(* PLC project CoDeSys External Library Template, WAGO e!COCKPIT e!COCKPIT, author 3S - Smart Software Solutions GmbH *)
(* stored: creationDateTime 2019-10-29T12:22:40.6298767, version 3.5.5.30, modificationDateTime 2019-10-24T14:40:07.960949, organization 3S - Smart Software Solutions GmbH *)
(* Library project template with all possible element types, docu and a sample project structure *)

FUNCTION_BLOCK fbFiltrWartoscAnalogowa
  VAR_INPUT
    rWartoscWejsciowa : REAL;
    rWartoscWejsciowaZaraportowana : REAL;
    rDeadband : REAL;
    tCzasMinimalny : TIME := TIME#5s0ms;
    tCzasMaksymalny : TIME := TIME#1m0s0ms;
    rWynikMnoznik : REAL := 1;
    rWynikOffset : REAL := 0;
  END_VAR
  VAR_OUTPUT
    rWartoscWyjsciowa : REAL;
  END_VAR
  VAR
    rWartoscWejsciowaZaraportowanaReferencja : REAL;
    fbCzasMinimalny : TON;
    fbCzasMaksymalny : TON;
    xCzasMinimalny : BOOL;
    xCzasMaksymalny : BOOL;
  END_VAR

            xCzasMinimalny := TRUE;
xCzasMaksymalny := TRUE;	

IF rWartoscWejsciowaZaraportowana <> rWartoscWejsciowaZaraportowanaReferencja THEN
	rWartoscWejsciowaZaraportowanaReferencja := rWartoscWejsciowaZaraportowana;
	xCzasMinimalny := FALSE;
	xCzasMaksymalny := FALSE;	
END_IF

IF fbCzasMinimalny.Q AND ABS(rWartoscWyjsciowa - (rWartoscWejsciowa * rWynikMnoznik + rWynikOffset)) > rDeadband THEN
	rWartoscWyjsciowa := rWartoscWejsciowa * rWynikMnoznik + rWynikOffset;
	xCzasMinimalny := FALSE;
	xCzasMaksymalny := FALSE;
END_IF

IF fbCzasMaksymalny.Q AND rWartoscWyjsciowa <> rWartoscWejsciowa * rWynikMnoznik + rWynikOffset THEN
	rWartoscWyjsciowa := rWartoscWejsciowa * rWynikMnoznik + rWynikOffset;
	xCzasMinimalny := FALSE;
	xCzasMaksymalny := FALSE;
END_IF

fbCzasMinimalny(IN := xCzasMinimalny, PT := tCzasMinimalny);
fbCzasMaksymalny(IN := xCzasMaksymalny , PT := tCzasMaksymalny);
          
END_FUNCTION_BLOCK
